// TIA Portal V19 export
DATA_BLOCK "Hmi"   // DB4
// stored: MemoryReserve 100
   VAR
      mainHeader : "LAF_typeHeader";   // Input from the status bar of the HMI
      operationInterlock : "LAF_typeOperationInterlockInterface";
   END_VAR
BEGIN
   mainHeader.plcToHmi.specialFunctionButtons.visibility := 16#7;
   mainHeader.plcToHmi.specialFunctionButtons.operatorControlAllowed := 16#F;
END_DATA_BLOCK
